{attribute 'GeneratedUsingTerminal: EL1502--0000'}
{attribute addProperty BoxType "EL1502--0000"}
{attribute addProperty Id "Output_functions_enabledAT %I*BOOL1Status_of_outputAT %I*BOOL1Set_counter_doneAT %I*BOOL1Counter_inhibitedAT %I*BOOL1Status_of_input_UDAT %I*BOOL1Status_of_input_clockAT %I*BOOL1TxPDO_ToggleAT %I*BOOL1Counter_valueAT %I*UDINT4"}
{attribute addProperty CRC "2101646797"}
{attribute addProperty Size "11"}
TYPE CNT_Inputs_7D4495CD :
STRUCT
	{attribute addProperty Name "Output_functions_enabled"}
	Output_functions_enabled AT %I* : BOOL;
	{attribute addProperty Name "Status_of_output"}
	Status_of_output AT %I* : BOOL;
	{attribute addProperty Name "Set_counter_done"}
	Set_counter_done AT %I* : BOOL;
	{attribute addProperty Name "Counter_inhibited"}
	Counter_inhibited AT %I* : BOOL;
	{attribute addProperty Name "Status_of_input_UD"}
	Status_of_input_UD AT %I* : BOOL;
	{attribute addProperty Name "Status_of_input_clock"}
	Status_of_input_clock AT %I* : BOOL;
	{attribute addProperty Name "TxPDO_Toggle"}
	TxPDO_Toggle AT %I* : BOOL;
	{attribute addProperty Name "Counter_value"}
	Counter_value AT %I* : UDINT;
END_STRUCT
END_TYPE

(* stored: Version 1.2.0.0, ProductVersion 3.1.4024.9
   DUT CNT_Inputs_7D4495CD: Id {165394e8-860a-4785-ac50-50849ea45697} *)
